// TIA Portal V21 export
FUNCTION "MODE SELECTION" : Void   // FC5, LAD
{ S7_Optimized_Access := 'TRUE' }
// stored: SetENOAutomatically false
   VAR_TEMP   // added for the SCL form of the ladder/FBD networks
      _w1 : Bool;
      _w2 : Bool;
      _w3 : Bool;
   END_VAR
BEGIN

REGION Network 1: MODE SELECTION
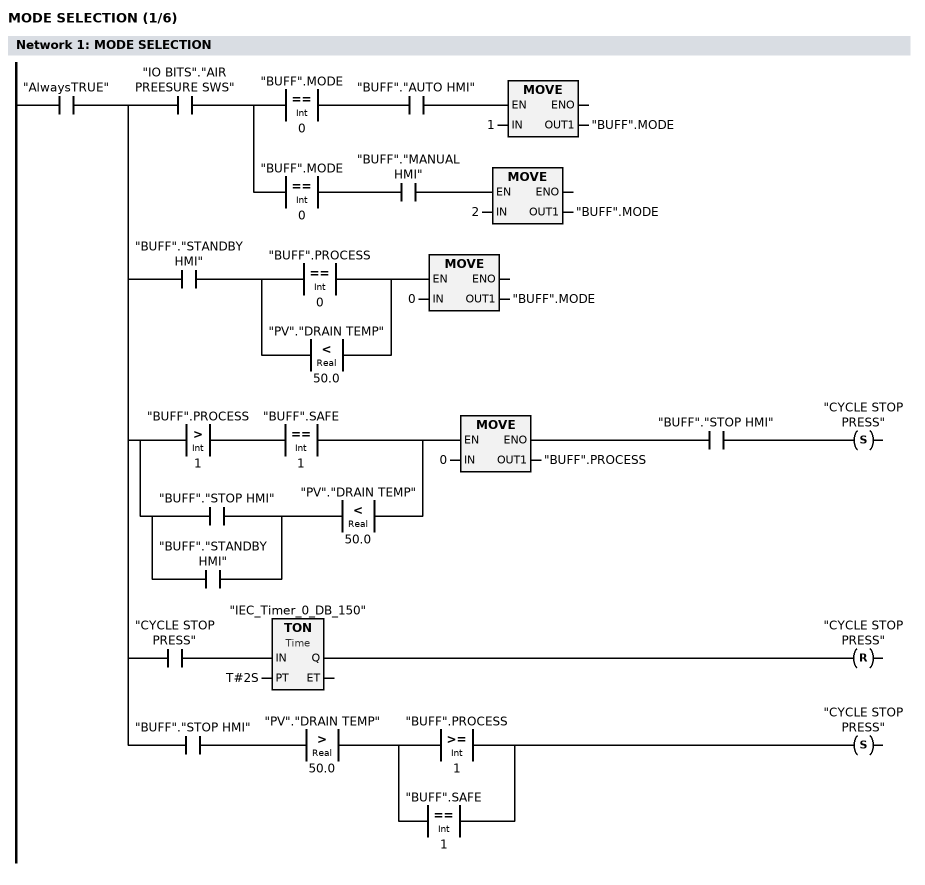
   RUNG wire#powerrail
      Contact( "AlwaysTRUE" )
      wire#w1
      Contact( "IO BITS"."AIR PREESURE SWS" )
      wire#w2
      { S7_Templates := "SrcType := Int" } EQ_Contact(in1 := "BUFF".MODE, in2 := 0)
      Contact( "BUFF"."AUTO HMI" )
      Move(in := 1, out1 => "BUFF".MODE)
   END_RUNG
   RUNG wire#w2
      { S7_Templates := "SrcType := Int" } EQ_Contact(in1 := "BUFF".MODE, in2 := 0)
      Contact( "BUFF"."MANUAL HMI" )
      Move(in := 2, out1 => "BUFF".MODE)
   END_RUNG
   RUNG wire#w1
      Contact( "BUFF"."STANDBY HMI" )
      wire#w3
      { S7_Templates := "SrcType := Int" } EQ_Contact(in1 := "BUFF".PROCESS, in2 := 0)
      wire#w4
      Move(in := 0, out1 => "BUFF".MODE)
   END_RUNG
   RUNG wire#w3
      { S7_Templates := "SrcType := Real" } LT_Contact(in1 := "PV"."DRAIN TEMP", in2 := 50.0)
   END_RUNG wire#w4
   RUNG wire#w1
      { S7_Templates := "SrcType := Int" } GT_Contact(in1 := "BUFF".PROCESS, in2 := 1)
      { S7_Templates := "SrcType := Int" } EQ_Contact(in1 := "BUFF".SAFE, in2 := 1)
      wire#w5
      Move(in := 0, out1 => "BUFF".PROCESS)
      Contact( "BUFF"."STOP HMI" )
      S_Coil( "CYCLE STOP PRESS" )
   END_RUNG
   RUNG wire#w1
      Contact( "BUFF"."STOP HMI" )
      wire#w6
      { S7_Templates := "SrcType := Real" } LT_Contact(in1 := "PV"."DRAIN TEMP", in2 := 50.0)
   END_RUNG wire#w5
   RUNG wire#w1
      Contact( "BUFF"."STANDBY HMI" )
   END_RUNG wire#w6
   RUNG wire#w1
      Contact( "CYCLE STOP PRESS" )
      { S7_Templates := "time_type := Time" } "IEC_Timer_0_DB_150".TON(pt := T#2S, et =>)
      R_Coil( "CYCLE STOP PRESS" )
   END_RUNG
   RUNG wire#w1
      Contact( "BUFF"."STOP HMI" )
      { S7_Templates := "SrcType := Real" } GT_Contact(in1 := "PV"."DRAIN TEMP", in2 := 50.0)
      wire#w7
      { S7_Templates := "SrcType := Int" } GE_Contact(in1 := "BUFF".PROCESS, in2 := 1)
      wire#w8
      S_Coil( "CYCLE STOP PRESS" )
   END_RUNG
   RUNG wire#w7
      { S7_Templates := "SrcType := Int" } EQ_Contact(in1 := "BUFF".SAFE, in2 := 1)
   END_RUNG wire#w8
   // the same network as SCL:
   #_w1 := "AlwaysTRUE" AND "IO BITS"."AIR PREESURE SWS";
   IF #_w1 AND ("BUFF".MODE = 0) AND "BUFF"."AUTO HMI" THEN "BUFF".MODE := 1; END_IF;
   IF #_w1 AND ("BUFF".MODE = 0) AND "BUFF"."MANUAL HMI" THEN "BUFF".MODE := 2; END_IF;
   IF "AlwaysTRUE" AND "BUFF"."STANDBY HMI" AND (("BUFF".PROCESS = 0) OR ("PV"."DRAIN TEMP" < 50.0)) THEN
       "BUFF".MODE := 0;
   END_IF;
   #_w2 := "AlwaysTRUE" AND ((("BUFF".PROCESS > 1) AND ("BUFF".SAFE = 1)) OR (("BUFF"."STOP HMI" OR "BUFF"."STANDBY HMI") AND ("PV"."DRAIN TEMP" < 50.0)));
   IF #_w2 THEN "BUFF".PROCESS := 0; END_IF;
   IF #_w2 AND "BUFF"."STOP HMI" THEN "CYCLE STOP PRESS" := TRUE; END_IF;
   "IEC_Timer_0_DB_150".TON(IN := "AlwaysTRUE" AND "CYCLE STOP PRESS", PT := T#2S);
   IF "IEC_Timer_0_DB_150".Q THEN "CYCLE STOP PRESS" := FALSE; END_IF;
   IF "AlwaysTRUE" AND "BUFF"."STOP HMI" AND ("PV"."DRAIN TEMP" > 50.0) AND (("BUFF".PROCESS >= 1) OR ("BUFF".SAFE = 1)) THEN
       "CYCLE STOP PRESS" := TRUE;
   END_IF;
END_REGION

REGION Network 2: PROCESS SELECTION
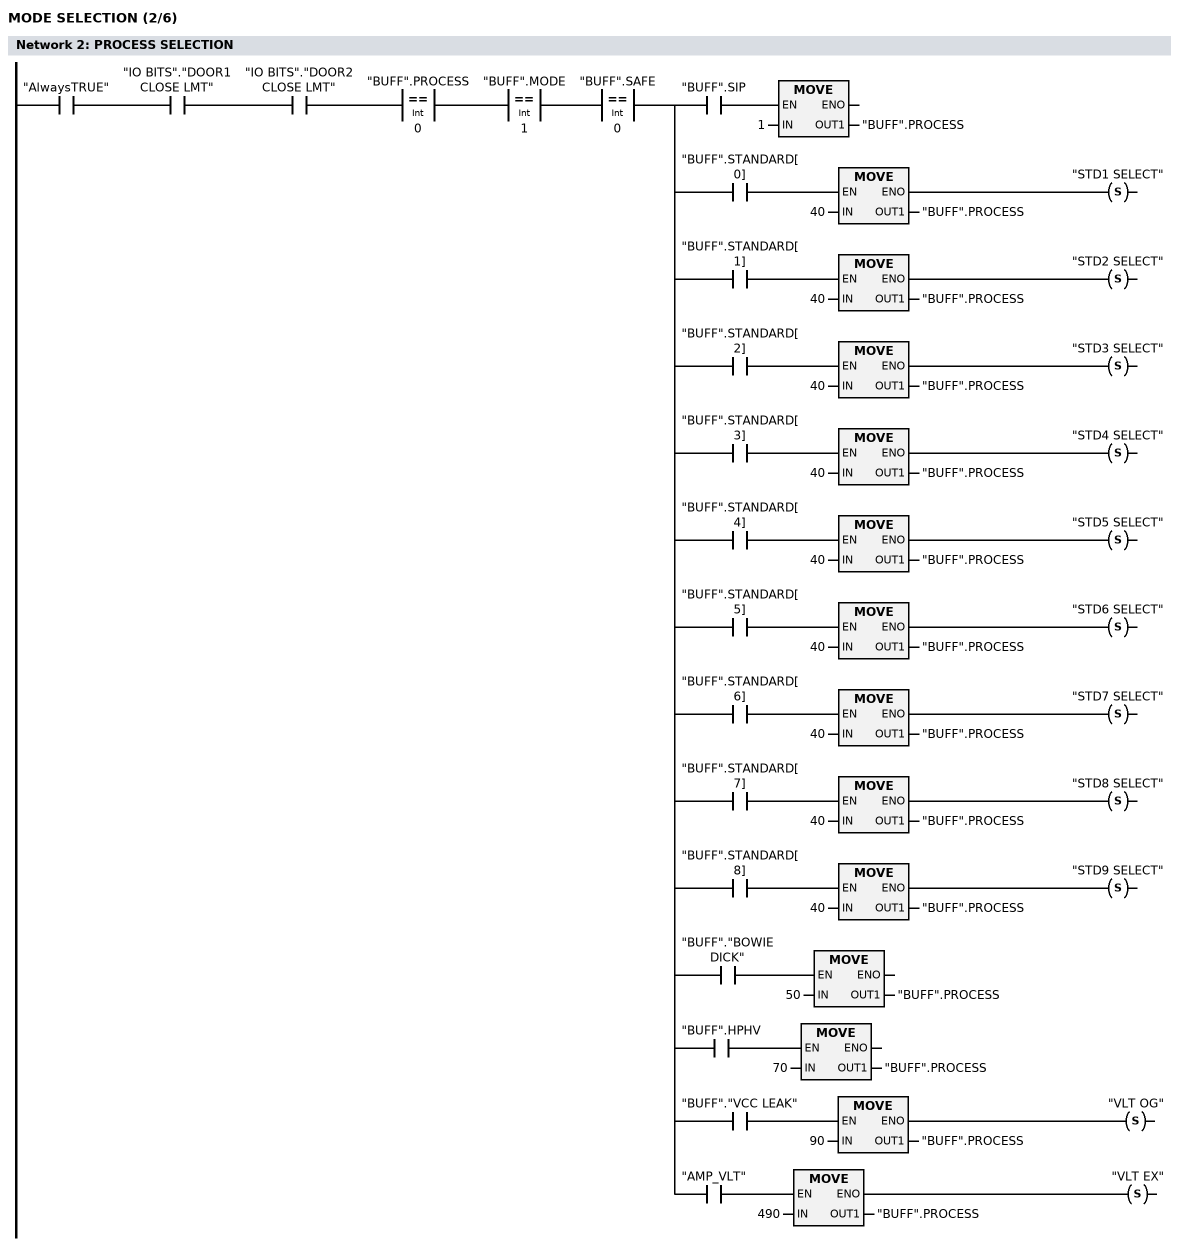
   RUNG wire#powerrail
      Contact( "AlwaysTRUE" )
      Contact( "IO BITS"."DOOR1 CLOSE LMT" )
      Contact( "IO BITS"."DOOR2 CLOSE LMT" )
      { S7_Templates := "SrcType := Int" } EQ_Contact(in1 := "BUFF".PROCESS, in2 := 0)
      { S7_Templates := "SrcType := Int" } EQ_Contact(in1 := "BUFF".MODE, in2 := 1)
      { S7_Templates := "SrcType := Int" } EQ_Contact(in1 := "BUFF".SAFE, in2 := 0)
      wire#w1
      Contact( "BUFF".SIP )
      Move(in := 1, out1 => "BUFF".PROCESS)
   END_RUNG
   RUNG wire#w1
      Contact( "BUFF".STANDARD[0] )
      Move(in := 40, out1 => "BUFF".PROCESS)
      S_Coil( "STD1 SELECT" )
   END_RUNG
   RUNG wire#w1
      Contact( "BUFF".STANDARD[1] )
      Move(in := 40, out1 => "BUFF".PROCESS)
      S_Coil( "STD2 SELECT" )
   END_RUNG
   RUNG wire#w1
      Contact( "BUFF".STANDARD[2] )
      Move(in := 40, out1 => "BUFF".PROCESS)
      S_Coil( "STD3 SELECT" )
   END_RUNG
   RUNG wire#w1
      Contact( "BUFF".STANDARD[3] )
      Move(in := 40, out1 => "BUFF".PROCESS)
      S_Coil( "STD4 SELECT" )
   END_RUNG
   RUNG wire#w1
      Contact( "BUFF".STANDARD[4] )
      Move(in := 40, out1 => "BUFF".PROCESS)
      S_Coil( "STD5 SELECT" )
   END_RUNG
   RUNG wire#w1
      Contact( "BUFF".STANDARD[5] )
      Move(in := 40, out1 => "BUFF".PROCESS)
      S_Coil( "STD6 SELECT" )
   END_RUNG
   RUNG wire#w1
      Contact( "BUFF".STANDARD[6] )
      Move(in := 40, out1 => "BUFF".PROCESS)
      S_Coil( "STD7 SELECT" )
   END_RUNG
   RUNG wire#w1
      Contact( "BUFF".STANDARD[7] )
      Move(in := 40, out1 => "BUFF".PROCESS)
      S_Coil( "STD8 SELECT" )
   END_RUNG
   RUNG wire#w1
      Contact( "BUFF".STANDARD[8] )
      Move(in := 40, out1 => "BUFF".PROCESS)
      S_Coil( "STD9 SELECT" )
   END_RUNG
   RUNG wire#w1
      Contact( "BUFF"."BOWIE DICK" )
      Move(in := 50, out1 => "BUFF".PROCESS)
   END_RUNG
   RUNG wire#w1
      Contact( "BUFF".HPHV )
      Move(in := 70, out1 => "BUFF".PROCESS)
   END_RUNG
   RUNG wire#w1
      Contact( "BUFF"."VCC LEAK" )
      Move(in := 90, out1 => "BUFF".PROCESS)
      S_Coil( "VLT OG" )
   END_RUNG
   RUNG wire#w1
      Contact( "AMP_VLT" )
      Move(in := 490, out1 => "BUFF".PROCESS)
      S_Coil( "VLT EX" )
   END_RUNG
   // the same network as SCL:
   #_w1 := "AlwaysTRUE" AND "IO BITS"."DOOR1 CLOSE LMT" AND "IO BITS"."DOOR2 CLOSE LMT" AND ("BUFF".PROCESS = 0) AND ("BUFF".MODE = 1) AND ("BUFF".SAFE = 0);
   IF #_w1 AND "BUFF".SIP THEN "BUFF".PROCESS := 1; END_IF;
   IF #_w1 AND "BUFF".STANDARD[0] THEN
       "BUFF".PROCESS := 40;
       "STD1 SELECT" := TRUE;
   END_IF;
   IF #_w1 AND "BUFF".STANDARD[1] THEN
       "BUFF".PROCESS := 40;
       "STD2 SELECT" := TRUE;
   END_IF;
   IF #_w1 AND "BUFF".STANDARD[2] THEN
       "BUFF".PROCESS := 40;
       "STD3 SELECT" := TRUE;
   END_IF;
   IF #_w1 AND "BUFF".STANDARD[3] THEN
       "BUFF".PROCESS := 40;
       "STD4 SELECT" := TRUE;
   END_IF;
   IF #_w1 AND "BUFF".STANDARD[4] THEN
       "BUFF".PROCESS := 40;
       "STD5 SELECT" := TRUE;
   END_IF;
   IF #_w1 AND "BUFF".STANDARD[5] THEN
       "BUFF".PROCESS := 40;
       "STD6 SELECT" := TRUE;
   END_IF;
   IF #_w1 AND "BUFF".STANDARD[6] THEN
       "BUFF".PROCESS := 40;
       "STD7 SELECT" := TRUE;
   END_IF;
   IF #_w1 AND "BUFF".STANDARD[7] THEN
       "BUFF".PROCESS := 40;
       "STD8 SELECT" := TRUE;
   END_IF;
   IF #_w1 AND "BUFF".STANDARD[8] THEN
       "BUFF".PROCESS := 40;
       "STD9 SELECT" := TRUE;
   END_IF;
   IF #_w1 AND "BUFF"."BOWIE DICK" THEN "BUFF".PROCESS := 50; END_IF;
   IF #_w1 AND "BUFF".HPHV THEN "BUFF".PROCESS := 70; END_IF;
   IF #_w1 AND "BUFF"."VCC LEAK" THEN
       "BUFF".PROCESS := 90;
       "VLT OG" := TRUE;
   END_IF;
   IF #_w1 AND "AMP_VLT" THEN
       "BUFF".PROCESS := 490;
       "VLT EX" := TRUE;
   END_IF;
END_REGION

REGION Network 3: DOOR OPERATION START
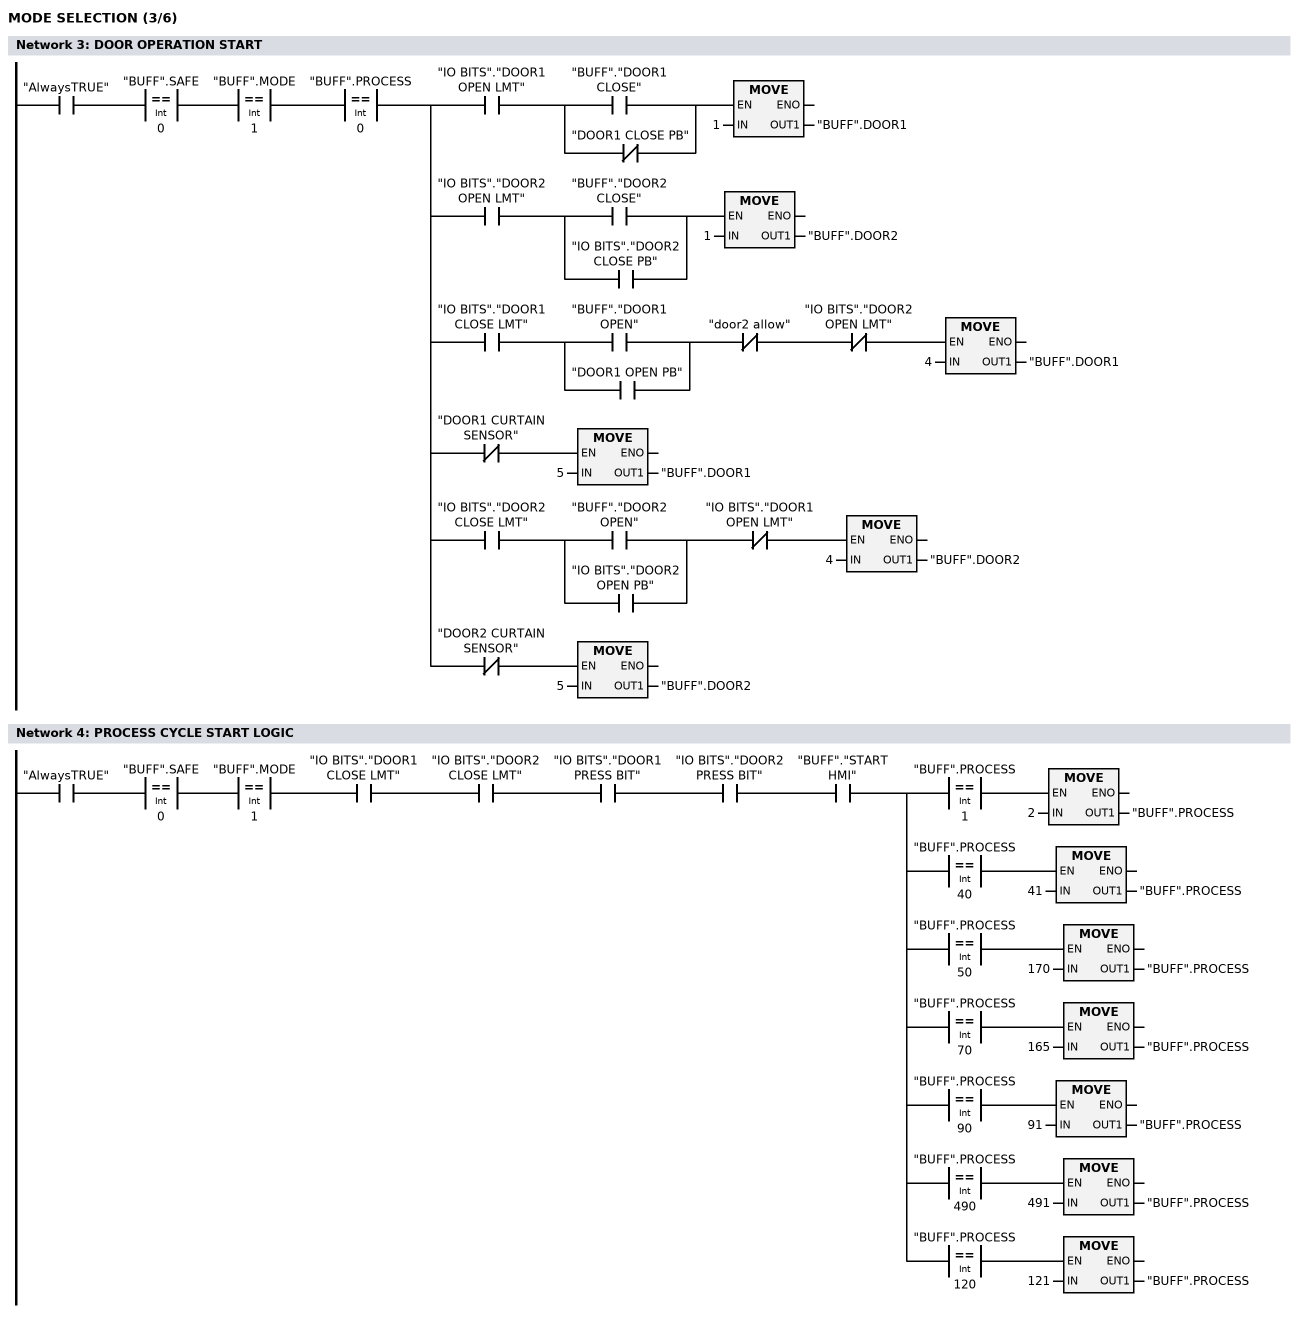
   RUNG wire#powerrail
      Contact( "AlwaysTRUE" )
      { S7_Templates := "SrcType := Int" } EQ_Contact(in1 := "BUFF".SAFE, in2 := 0)
      { S7_Templates := "SrcType := Int" } EQ_Contact(in1 := "BUFF".MODE, in2 := 1)
      { S7_Templates := "SrcType := Int" } EQ_Contact(in1 := "BUFF".PROCESS, in2 := 0)
      wire#w1
      Contact( "IO BITS"."DOOR1 OPEN LMT" )
      wire#w2
      Contact( "BUFF"."DOOR1 CLOSE" )
      wire#w3
      Move(in := 1, out1 => "BUFF".DOOR1)
   END_RUNG
   RUNG wire#w2
      I_Contact( "DOOR1 CLOSE PB" )
   END_RUNG wire#w3
   RUNG wire#w1
      Contact( "IO BITS"."DOOR2 OPEN LMT" )
      wire#w4
      Contact( "BUFF"."DOOR2 CLOSE" )
      wire#w5
      Move(in := 1, out1 => "BUFF".DOOR2)
   END_RUNG
   RUNG wire#w4
      Contact( "IO BITS"."DOOR2 CLOSE PB" )
   END_RUNG wire#w5
   RUNG wire#w1
      Contact( "IO BITS"."DOOR1 CLOSE LMT" )
      wire#w6
      Contact( "BUFF"."DOOR1 OPEN" )
      wire#w7
      I_Contact( "door2 allow" )
      I_Contact( "IO BITS"."DOOR2 OPEN LMT" )
      Move(in := 4, out1 => "BUFF".DOOR1)
   END_RUNG
   RUNG wire#w6
      Contact( "DOOR1 OPEN PB" )
   END_RUNG wire#w7
   RUNG wire#w1
      I_Contact( "DOOR1 CURTAIN SENSOR" )
      Move(in := 5, out1 => "BUFF".DOOR1)
   END_RUNG
   RUNG wire#w1
      Contact( "IO BITS"."DOOR2 CLOSE LMT" )
      wire#w8
      Contact( "BUFF"."DOOR2 OPEN" )
      wire#w9
      I_Contact( "IO BITS"."DOOR1 OPEN LMT" )
      Move(in := 4, out1 => "BUFF".DOOR2)
   END_RUNG
   RUNG wire#w8
      Contact( "IO BITS"."DOOR2 OPEN PB" )
   END_RUNG wire#w9
   RUNG wire#w1
      I_Contact( "DOOR2 CURTAIN SENSOR" )
      Move(in := 5, out1 => "BUFF".DOOR2)
   END_RUNG
   // the same network as SCL:
   #_w1 := "AlwaysTRUE" AND ("BUFF".SAFE = 0) AND ("BUFF".MODE = 1) AND ("BUFF".PROCESS = 0);
   IF #_w1 AND "IO BITS"."DOOR1 OPEN LMT" AND ("BUFF"."DOOR1 CLOSE" OR NOT "DOOR1 CLOSE PB") THEN
       "BUFF".DOOR1 := 1;
   END_IF;
   IF #_w1 AND "IO BITS"."DOOR2 OPEN LMT" AND ("BUFF"."DOOR2 CLOSE" OR "IO BITS"."DOOR2 CLOSE PB") THEN
       "BUFF".DOOR2 := 1;
   END_IF;
   IF #_w1 AND "IO BITS"."DOOR1 CLOSE LMT" AND ("BUFF"."DOOR1 OPEN" OR "DOOR1 OPEN PB") AND NOT "door2 allow" AND NOT "IO BITS"."DOOR2 OPEN LMT" THEN
       "BUFF".DOOR1 := 4;
   END_IF;
   IF #_w1 AND NOT "DOOR1 CURTAIN SENSOR" THEN "BUFF".DOOR1 := 5; END_IF;
   IF #_w1 AND "IO BITS"."DOOR2 CLOSE LMT" AND ("BUFF"."DOOR2 OPEN" OR "IO BITS"."DOOR2 OPEN PB") AND NOT "IO BITS"."DOOR1 OPEN LMT" THEN
       "BUFF".DOOR2 := 4;
   END_IF;
   IF #_w1 AND NOT "DOOR2 CURTAIN SENSOR" THEN "BUFF".DOOR2 := 5; END_IF;
END_REGION

REGION Network 4: PROCESS CYCLE START LOGIC
   RUNG wire#powerrail
      Contact( "AlwaysTRUE" )
      { S7_Templates := "SrcType := Int" } EQ_Contact(in1 := "BUFF".SAFE, in2 := 0)
      { S7_Templates := "SrcType := Int" } EQ_Contact(in1 := "BUFF".MODE, in2 := 1)
      Contact( "IO BITS"."DOOR1 CLOSE LMT" )
      Contact( "IO BITS"."DOOR2 CLOSE LMT" )
      Contact( "IO BITS"."DOOR1 PRESS BIT" )
      Contact( "IO BITS"."DOOR2 PRESS BIT" )
      Contact( "BUFF"."START HMI" )
      wire#w1
      { S7_Templates := "SrcType := Int" } EQ_Contact(in1 := "BUFF".PROCESS, in2 := 1)
      Move(in := 2, out1 => "BUFF".PROCESS)
   END_RUNG
   RUNG wire#w1
      { S7_Templates := "SrcType := Int" } EQ_Contact(in1 := "BUFF".PROCESS, in2 := 40)
      Move(in := 41, out1 => "BUFF".PROCESS)
   END_RUNG
   RUNG wire#w1
      { S7_Templates := "SrcType := Int" } EQ_Contact(in1 := "BUFF".PROCESS, in2 := 50)
      Move(in := 170, out1 => "BUFF".PROCESS)
   END_RUNG
   RUNG wire#w1
      { S7_Templates := "SrcType := Int" } EQ_Contact(in1 := "BUFF".PROCESS, in2 := 70)
      Move(in := 165, out1 => "BUFF".PROCESS)
   END_RUNG
   RUNG wire#w1
      { S7_Templates := "SrcType := Int" } EQ_Contact(in1 := "BUFF".PROCESS, in2 := 90)
      Move(in := 91, out1 => "BUFF".PROCESS)
   END_RUNG
   RUNG wire#w1
      { S7_Templates := "SrcType := Int" } EQ_Contact(in1 := "BUFF".PROCESS, in2 := 490)
      Move(in := 491, out1 => "BUFF".PROCESS)
   END_RUNG
   RUNG wire#w1
      { S7_Templates := "SrcType := Int" } EQ_Contact(in1 := "BUFF".PROCESS, in2 := 120)
      Move(in := 121, out1 => "BUFF".PROCESS)
   END_RUNG
   // the same network as SCL:
   #_w1 := "AlwaysTRUE" AND ("BUFF".SAFE = 0) AND ("BUFF".MODE = 1) AND "IO BITS"."DOOR1 CLOSE LMT" AND "IO BITS"."DOOR2 CLOSE LMT" AND "IO BITS"."DOOR1 PRESS BIT" AND "IO BITS"."DOOR2 PRESS BIT" AND "BUFF"."START HMI";
   IF #_w1 AND ("BUFF".PROCESS = 1) THEN "BUFF".PROCESS := 2; END_IF;
   IF #_w1 AND ("BUFF".PROCESS = 40) THEN "BUFF".PROCESS := 41; END_IF;
   IF #_w1 AND ("BUFF".PROCESS = 50) THEN "BUFF".PROCESS := 170; END_IF;
   IF #_w1 AND ("BUFF".PROCESS = 70) THEN "BUFF".PROCESS := 165; END_IF;
   IF #_w1 AND ("BUFF".PROCESS = 90) THEN "BUFF".PROCESS := 91; END_IF;
   IF #_w1 AND ("BUFF".PROCESS = 490) THEN "BUFF".PROCESS := 491; END_IF;
   IF #_w1 AND ("BUFF".PROCESS = 120) THEN "BUFF".PROCESS := 121; END_IF;
END_REGION

REGION Network 5: DOOR CLOSE LOGIC
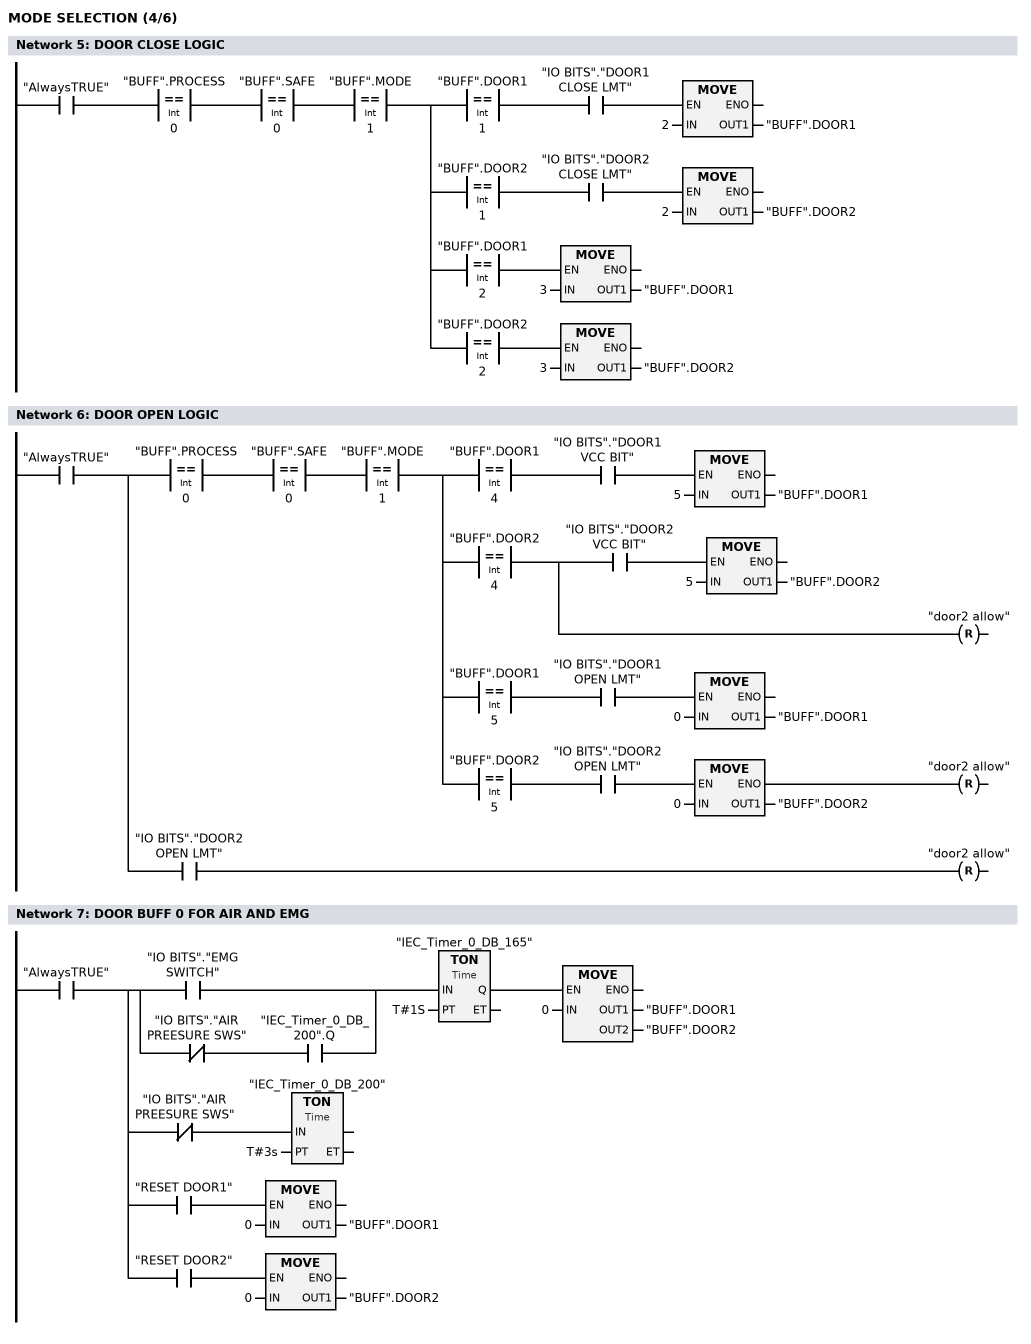
   RUNG wire#powerrail
      Contact( "AlwaysTRUE" )
      { S7_Templates := "SrcType := Int" } EQ_Contact(in1 := "BUFF".PROCESS, in2 := 0)
      { S7_Templates := "SrcType := Int" } EQ_Contact(in1 := "BUFF".SAFE, in2 := 0)
      { S7_Templates := "SrcType := Int" } EQ_Contact(in1 := "BUFF".MODE, in2 := 1)
      wire#w1
      { S7_Templates := "SrcType := Int" } EQ_Contact(in1 := "BUFF".DOOR1, in2 := 1)
      Contact( "IO BITS"."DOOR1 CLOSE LMT" )
      Move(in := 2, out1 => "BUFF".DOOR1)
   END_RUNG
   RUNG wire#w1
      { S7_Templates := "SrcType := Int" } EQ_Contact(in1 := "BUFF".DOOR2, in2 := 1)
      Contact( "IO BITS"."DOOR2 CLOSE LMT" )
      Move(in := 2, out1 => "BUFF".DOOR2)
   END_RUNG
   RUNG wire#w1
      { S7_Templates := "SrcType := Int" } EQ_Contact(in1 := "BUFF".DOOR1, in2 := 2)
      Move(in := 3, out1 => "BUFF".DOOR1)
   END_RUNG
   RUNG wire#w1
      { S7_Templates := "SrcType := Int" } EQ_Contact(in1 := "BUFF".DOOR2, in2 := 2)
      Move(in := 3, out1 => "BUFF".DOOR2)
   END_RUNG
   // the same network as SCL:
   #_w1 := "AlwaysTRUE" AND ("BUFF".PROCESS = 0) AND ("BUFF".SAFE = 0) AND ("BUFF".MODE = 1);
   IF #_w1 AND ("BUFF".DOOR1 = 1) AND "IO BITS"."DOOR1 CLOSE LMT" THEN "BUFF".DOOR1 := 2; END_IF;
   IF #_w1 AND ("BUFF".DOOR2 = 1) AND "IO BITS"."DOOR2 CLOSE LMT" THEN "BUFF".DOOR2 := 2; END_IF;
   IF #_w1 AND ("BUFF".DOOR1 = 2) THEN "BUFF".DOOR1 := 3; END_IF;
   IF #_w1 AND ("BUFF".DOOR2 = 2) THEN "BUFF".DOOR2 := 3; END_IF;
END_REGION

REGION Network 6: DOOR OPEN LOGIC
   RUNG wire#powerrail
      Contact( "AlwaysTRUE" )
      wire#w1
      { S7_Templates := "SrcType := Int" } EQ_Contact(in1 := "BUFF".PROCESS, in2 := 0)
      { S7_Templates := "SrcType := Int" } EQ_Contact(in1 := "BUFF".SAFE, in2 := 0)
      { S7_Templates := "SrcType := Int" } EQ_Contact(in1 := "BUFF".MODE, in2 := 1)
      wire#w2
      { S7_Templates := "SrcType := Int" } EQ_Contact(in1 := "BUFF".DOOR1, in2 := 4)
      Contact( "IO BITS"."DOOR1 VCC BIT" )
      Move(in := 5, out1 => "BUFF".DOOR1)
   END_RUNG
   RUNG wire#w2
      { S7_Templates := "SrcType := Int" } EQ_Contact(in1 := "BUFF".DOOR2, in2 := 4)
      wire#w3
      Contact( "IO BITS"."DOOR2 VCC BIT" )
      Move(in := 5, out1 => "BUFF".DOOR2)
   END_RUNG
   RUNG wire#w3
      R_Coil( "door2 allow" )
   END_RUNG
   RUNG wire#w2
      { S7_Templates := "SrcType := Int" } EQ_Contact(in1 := "BUFF".DOOR1, in2 := 5)
      Contact( "IO BITS"."DOOR1 OPEN LMT" )
      Move(in := 0, out1 => "BUFF".DOOR1)
   END_RUNG
   RUNG wire#w2
      { S7_Templates := "SrcType := Int" } EQ_Contact(in1 := "BUFF".DOOR2, in2 := 5)
      Contact( "IO BITS"."DOOR2 OPEN LMT" )
      Move(in := 0, out1 => "BUFF".DOOR2)
      R_Coil( "door2 allow" )
   END_RUNG
   RUNG wire#w1
      Contact( "IO BITS"."DOOR2 OPEN LMT" )
      R_Coil( "door2 allow" )
   END_RUNG
   // the same network as SCL:
   #_w1 := "AlwaysTRUE" AND ("BUFF".PROCESS = 0) AND ("BUFF".SAFE = 0) AND ("BUFF".MODE = 1);
   IF #_w1 AND ("BUFF".DOOR1 = 4) AND "IO BITS"."DOOR1 VCC BIT" THEN "BUFF".DOOR1 := 5; END_IF;
   #_w2 := #_w1 AND ("BUFF".DOOR2 = 4);
   IF #_w2 AND "IO BITS"."DOOR2 VCC BIT" THEN "BUFF".DOOR2 := 5; END_IF;
   IF #_w2 THEN "door2 allow" := FALSE; END_IF;
   IF #_w1 AND ("BUFF".DOOR1 = 5) AND "IO BITS"."DOOR1 OPEN LMT" THEN "BUFF".DOOR1 := 0; END_IF;
   #_w3 := #_w1 AND ("BUFF".DOOR2 = 5) AND "IO BITS"."DOOR2 OPEN LMT";
   IF #_w3 THEN
       "BUFF".DOOR2 := 0;
       "door2 allow" := FALSE;
   END_IF;
   IF "AlwaysTRUE" AND "IO BITS"."DOOR2 OPEN LMT" THEN "door2 allow" := FALSE; END_IF;
END_REGION

REGION Network 7: DOOR BUFF 0 FOR AIR AND EMG
   RUNG wire#powerrail
      Contact( "AlwaysTRUE" )
      wire#w1
      Contact( "IO BITS"."EMG SWITCH" )
      wire#w2
      { S7_Templates := "time_type := Time" } "IEC_Timer_0_DB_165".TON(pt := T#1S, et =>)
      Move(in := 0, out1 => "BUFF".DOOR1, out2 => "BUFF".DOOR2)
   END_RUNG
   RUNG wire#w1
      I_Contact( "IO BITS"."AIR PREESURE SWS" )
      Contact( "IEC_Timer_0_DB_200".Q )
   END_RUNG wire#w2
   RUNG wire#w1
      I_Contact( "IO BITS"."AIR PREESURE SWS" )
      { S7_Templates := "time_type := Time" } "IEC_Timer_0_DB_200".TON(pt := T#3s, et =>)
   END_RUNG
   RUNG wire#w1
      Contact( "RESET DOOR1" )
      Move(in := 0, out1 => "BUFF".DOOR1)
   END_RUNG
   RUNG wire#w1
      Contact( "RESET DOOR2" )
      Move(in := 0, out1 => "BUFF".DOOR2)
   END_RUNG
   // the same network as SCL:
   "IEC_Timer_0_DB_165".TON(IN := "AlwaysTRUE" AND ("IO BITS"."EMG SWITCH" OR (NOT "IO BITS"."AIR PREESURE SWS" AND "IEC_Timer_0_DB_200".Q)),
                           PT := T#1S);
   IF "IEC_Timer_0_DB_165".Q THEN
       "BUFF".DOOR1 := 0;
       "BUFF".DOOR2 := 0;
   END_IF;
   "IEC_Timer_0_DB_200".TON(IN := "AlwaysTRUE" AND NOT "IO BITS"."AIR PREESURE SWS", PT := T#3s);
   IF "AlwaysTRUE" AND "RESET DOOR1" THEN "BUFF".DOOR1 := 0; END_IF;
   IF "AlwaysTRUE" AND "RESET DOOR2" THEN "BUFF".DOOR2 := 0; END_IF;
END_REGION

REGION Network 8: MANUAL RESET
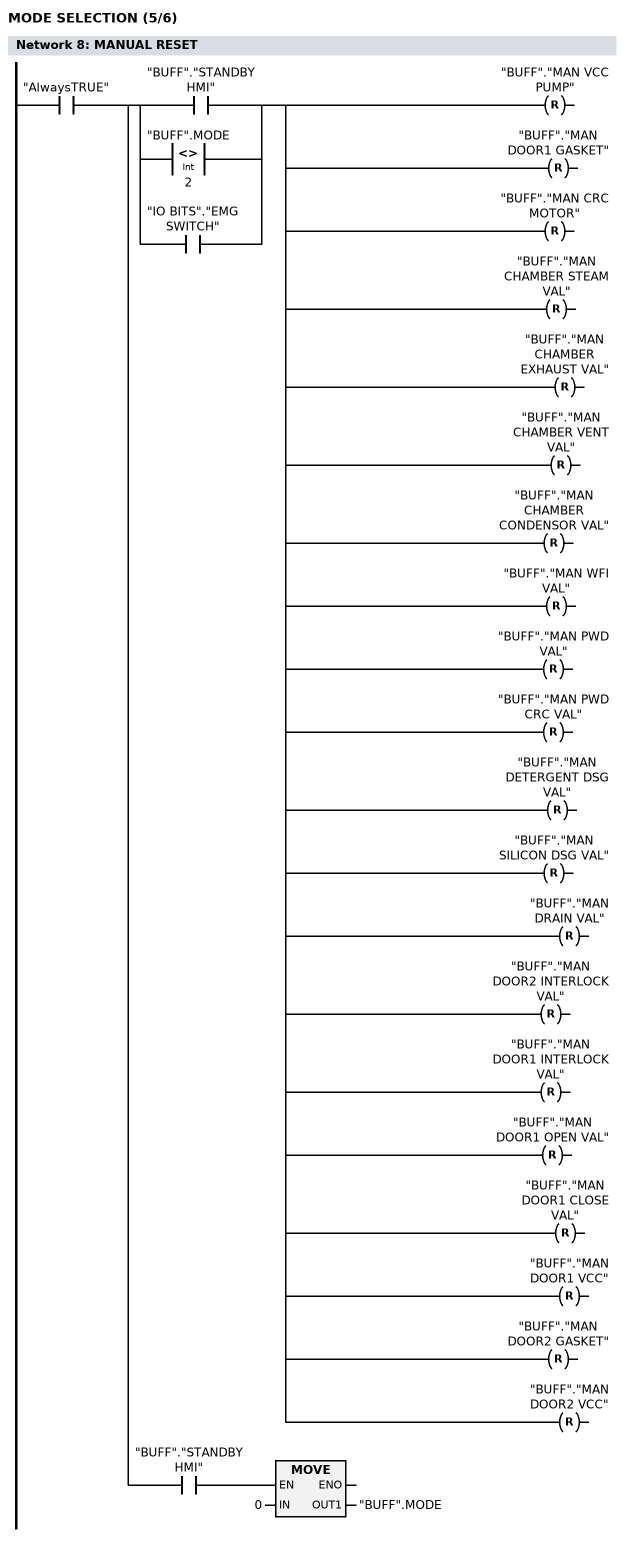
   RUNG wire#powerrail
      Contact( "AlwaysTRUE" )
      wire#w1
      Contact( "BUFF"."STANDBY HMI" )
      wire#w2
      R_Coil( "BUFF"."MAN VCC PUMP" )
   END_RUNG
   RUNG wire#w1
      { S7_Templates := "SrcType := Int" } NE_Contact(in1 := "BUFF".MODE, in2 := 2)
   END_RUNG wire#w2
   RUNG wire#w1
      Contact( "IO BITS"."EMG SWITCH" )
   END_RUNG wire#w2
   RUNG wire#w2
      R_Coil( "BUFF"."MAN DOOR1 GASKET" )
   END_RUNG
   RUNG wire#w2
      R_Coil( "BUFF"."MAN CRC MOTOR" )
   END_RUNG
   RUNG wire#w2
      R_Coil( "BUFF"."MAN CHAMBER STEAM VAL" )
   END_RUNG
   RUNG wire#w2
      R_Coil( "BUFF"."MAN CHAMBER EXHAUST VAL" )
   END_RUNG
   RUNG wire#w2
      R_Coil( "BUFF"."MAN CHAMBER VENT VAL" )
   END_RUNG
   RUNG wire#w2
      R_Coil( "BUFF"."MAN CHAMBER CONDENSOR VAL" )
   END_RUNG
   RUNG wire#w2
      R_Coil( "BUFF"."MAN WFI VAL" )
   END_RUNG
   RUNG wire#w2
      R_Coil( "BUFF"."MAN PWD VAL" )
   END_RUNG
   RUNG wire#w2
      R_Coil( "BUFF"."MAN PWD CRC VAL" )
   END_RUNG
   RUNG wire#w2
      R_Coil( "BUFF"."MAN DETERGENT DSG VAL" )
   END_RUNG
   RUNG wire#w2
      R_Coil( "BUFF"."MAN SILICON DSG VAL" )
   END_RUNG
   RUNG wire#w2
      R_Coil( "BUFF"."MAN DRAIN VAL" )
   END_RUNG
   RUNG wire#w2
      R_Coil( "BUFF"."MAN DOOR2 INTERLOCK VAL" )
   END_RUNG
   RUNG wire#w2
      R_Coil( "BUFF"."MAN DOOR1 INTERLOCK VAL" )
   END_RUNG
   RUNG wire#w2
      R_Coil( "BUFF"."MAN DOOR1 OPEN VAL" )
   END_RUNG
   RUNG wire#w2
      R_Coil( "BUFF"."MAN DOOR1 CLOSE VAL" )
   END_RUNG
   RUNG wire#w2
      R_Coil( "BUFF"."MAN DOOR1 VCC" )
   END_RUNG
   RUNG wire#w2
      R_Coil( "BUFF"."MAN DOOR2 GASKET" )
   END_RUNG
   RUNG wire#w2
      R_Coil( "BUFF"."MAN DOOR2 VCC" )
   END_RUNG
   RUNG wire#w1
      Contact( "BUFF"."STANDBY HMI" )
      Move(in := 0, out1 => "BUFF".MODE)
   END_RUNG
   // the same network as SCL:
   IF "AlwaysTRUE" AND ("BUFF"."STANDBY HMI" OR ("BUFF".MODE <> 2) OR "IO BITS"."EMG SWITCH") THEN
       "BUFF"."MAN VCC PUMP" := FALSE;
       "BUFF"."MAN DOOR1 GASKET" := FALSE;
       "BUFF"."MAN CRC MOTOR" := FALSE;
       "BUFF"."MAN CHAMBER STEAM VAL" := FALSE;
       "BUFF"."MAN CHAMBER EXHAUST VAL" := FALSE;
       "BUFF"."MAN CHAMBER VENT VAL" := FALSE;
       "BUFF"."MAN CHAMBER CONDENSOR VAL" := FALSE;
       "BUFF"."MAN WFI VAL" := FALSE;
       "BUFF"."MAN PWD VAL" := FALSE;
       "BUFF"."MAN PWD CRC VAL" := FALSE;
       "BUFF"."MAN DETERGENT DSG VAL" := FALSE;
       "BUFF"."MAN SILICON DSG VAL" := FALSE;
       "BUFF"."MAN DRAIN VAL" := FALSE;
       "BUFF"."MAN DOOR2 INTERLOCK VAL" := FALSE;
       "BUFF"."MAN DOOR1 INTERLOCK VAL" := FALSE;
       "BUFF"."MAN DOOR1 OPEN VAL" := FALSE;
       "BUFF"."MAN DOOR1 CLOSE VAL" := FALSE;
       "BUFF"."MAN DOOR1 VCC" := FALSE;
       "BUFF"."MAN DOOR2 GASKET" := FALSE;
       "BUFF"."MAN DOOR2 VCC" := FALSE;
   END_IF;
   IF "AlwaysTRUE" AND "BUFF"."STANDBY HMI" THEN "BUFF".MODE := 0; END_IF;
END_REGION

REGION Network 9
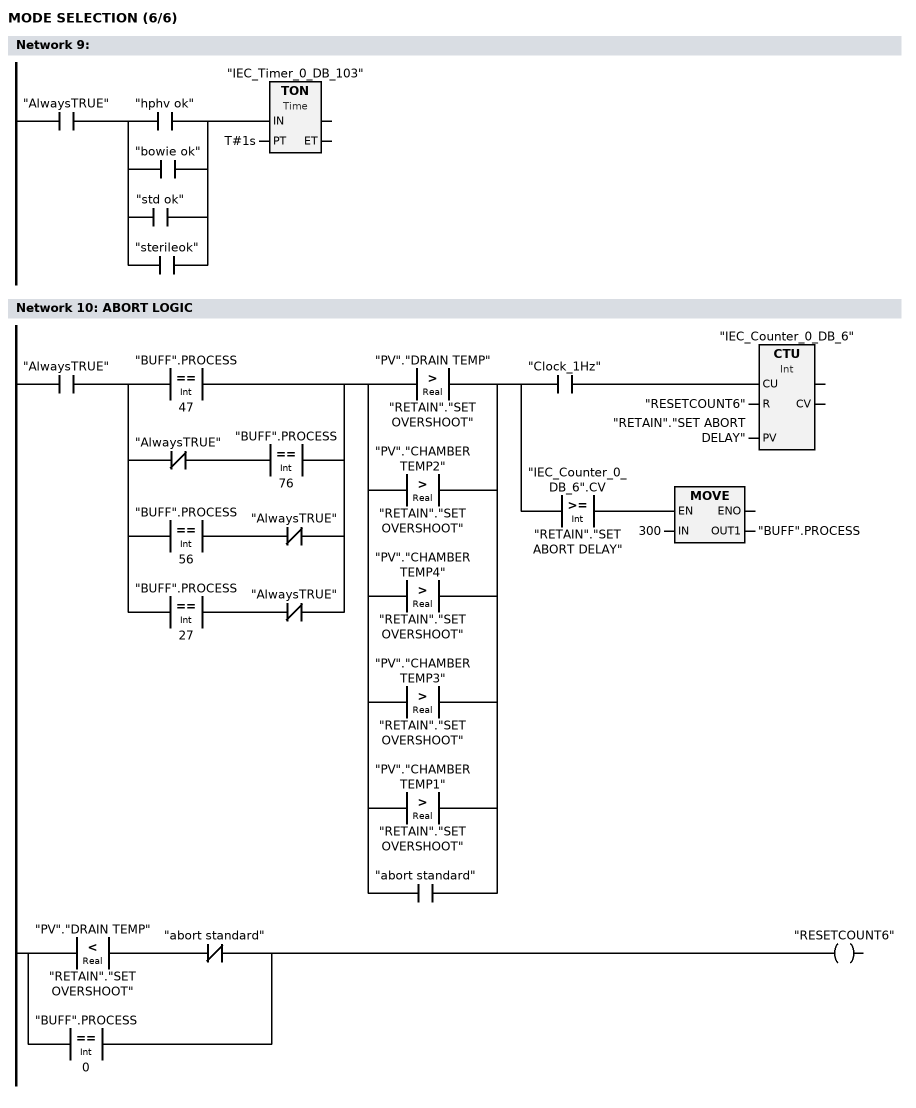
   RUNG wire#powerrail
      Contact( "AlwaysTRUE" )
      wire#w1
      Contact( "hphv ok" )
      wire#w2
      { S7_Templates := "time_type := Time" } "IEC_Timer_0_DB_103".TON(pt := T#1s, et =>)
   END_RUNG
   RUNG wire#w1
      Contact( "bowie ok" )
   END_RUNG wire#w2
   RUNG wire#w1
      Contact( "std ok" )
   END_RUNG wire#w2
   RUNG wire#w1
      Contact( "sterileok" )
   END_RUNG wire#w2
   // the same network as SCL:
   "IEC_Timer_0_DB_103".TON(IN := "AlwaysTRUE" AND ("hphv ok" OR "bowie ok" OR "std ok" OR "sterileok"),
                           PT := T#1s);
END_REGION

REGION Network 10: ABORT LOGIC
   RUNG wire#powerrail
      Contact( "AlwaysTRUE" )
      wire#w1
      { S7_Templates := "SrcType := Int" } EQ_Contact(in1 := "BUFF".PROCESS, in2 := 47)
      wire#w2
      { S7_Templates := "SrcType := Real" } GT_Contact(in1 := "PV"."DRAIN TEMP", in2 := "RETAIN"."SET OVERSHOOT")
      wire#w3
      Contact( "Clock_1Hz" )
      { S7_Templates := "value_type := Int" } "IEC_Counter_0_DB_6".CTU(r := "RESETCOUNT6", pv := "RETAIN"."SET ABORT DELAY", cv =>)
   END_RUNG
   RUNG wire#w1
      I_Contact( "AlwaysTRUE" )
      { S7_Templates := "SrcType := Int" } EQ_Contact(in1 := "BUFF".PROCESS, in2 := 76)
   END_RUNG wire#w2
   RUNG wire#w1
      { S7_Templates := "SrcType := Int" } EQ_Contact(in1 := "BUFF".PROCESS, in2 := 56)
      I_Contact( "AlwaysTRUE" )
   END_RUNG wire#w2
   RUNG wire#w1
      { S7_Templates := "SrcType := Int" } EQ_Contact(in1 := "BUFF".PROCESS, in2 := 27)
      I_Contact( "AlwaysTRUE" )
   END_RUNG wire#w2
   RUNG wire#w2
      { S7_Templates := "SrcType := Real" } GT_Contact(in1 := "PV"."CHAMBER TEMP2", in2 := "RETAIN"."SET OVERSHOOT")
   END_RUNG wire#w3
   RUNG wire#w2
      { S7_Templates := "SrcType := Real" } GT_Contact(in1 := "PV"."CHAMBER TEMP4", in2 := "RETAIN"."SET OVERSHOOT")
   END_RUNG wire#w3
   RUNG wire#w2
      { S7_Templates := "SrcType := Real" } GT_Contact(in1 := "PV"."CHAMBER TEMP3", in2 := "RETAIN"."SET OVERSHOOT")
   END_RUNG wire#w3
   RUNG wire#w2
      { S7_Templates := "SrcType := Real" } GT_Contact(in1 := "PV"."CHAMBER TEMP1", in2 := "RETAIN"."SET OVERSHOOT")
   END_RUNG wire#w3
   RUNG wire#w2
      Contact( "abort standard" )
   END_RUNG wire#w3
   RUNG wire#w3
      { S7_Templates := "SrcType := Int" } GE_Contact(in1 := "IEC_Counter_0_DB_6".CV, in2 := "RETAIN"."SET ABORT DELAY")
      Move(in := 300, out1 => "BUFF".PROCESS)
   END_RUNG
   RUNG wire#powerrail
      { S7_Templates := "SrcType := Real" } LT_Contact(in1 := "PV"."DRAIN TEMP", in2 := "RETAIN"."SET OVERSHOOT")
      I_Contact( "abort standard" )
      wire#w4
      Coil( "RESETCOUNT6" )
   END_RUNG
   RUNG wire#powerrail
      { S7_Templates := "SrcType := Int" } EQ_Contact(in1 := "BUFF".PROCESS, in2 := 0)
   END_RUNG wire#w4
   // the same network as SCL:
   #_w1 := "AlwaysTRUE" AND (("BUFF".PROCESS = 47) OR (NOT "AlwaysTRUE" AND ("BUFF".PROCESS = 76)) OR (("BUFF".PROCESS = 56) AND NOT "AlwaysTRUE") OR (("BUFF".PROCESS = 27) AND NOT "AlwaysTRUE")) AND (("PV"."DRAIN TEMP" > "RETAIN"."SET OVERSHOOT") OR ("PV"."CHAMBER TEMP2" > "RETAIN"."SET OVERSHOOT") OR ("PV"."CHAMBER TEMP4" > "RETAIN"."SET OVERSHOOT") OR ("PV"."CHAMBER TEMP3" > "RETAIN"."SET OVERSHOOT") OR ("PV"."CHAMBER TEMP1" > "RETAIN"."SET OVERSHOOT") OR "abort standard");
   "IEC_Counter_0_DB_6".CTU(CU := #_w1 AND "Clock_1Hz", R := "RESETCOUNT6", PV := "RETAIN"."SET ABORT DELAY");
   IF #_w1 AND ("IEC_Counter_0_DB_6".CV >= "RETAIN"."SET ABORT DELAY") THEN "BUFF".PROCESS := 300; END_IF;
   "RESETCOUNT6" := (("PV"."DRAIN TEMP" < "RETAIN"."SET OVERSHOOT") AND NOT "abort standard") OR ("BUFF".PROCESS = 0);
END_REGION
END_FUNCTION
